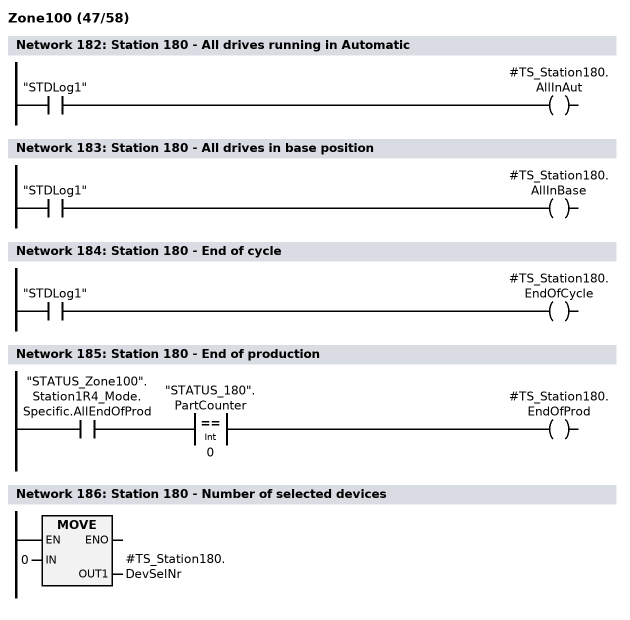
   RUNG wire#powerrail
      Contact( "STDLog1" )
      Coil( #TS_Station180.AllInAut )
   END_RUNG
   // the same network as SCL:
   #TS_Station180.AllInAut := "STDLog1";
END_REGION

REGION Network 183: Station 180 - All drives in base position
   RUNG wire#powerrail
      Contact( "STDLog1" )
      Coil( #TS_Station180.AllInBase )
   END_RUNG
   // the same network as SCL:
   #TS_Station180.AllInBase := "STDLog1";
END_REGION

REGION Network 184: Station 180 - End of cycle
   RUNG wire#powerrail
      Contact( "STDLog1" )
      Coil( #TS_Station180.EndOfCycle )
   END_RUNG
   // the same network as SCL:
   #TS_Station180.EndOfCycle := "STDLog1";
END_REGION

REGION Network 185: Station 180 - End of production
   RUNG wire#powerrail
      Contact( "STATUS_Zone100".Station1R4_Mode.Specific.AllEndOfProd )
      { S7_Templates := "SrcType := Int" } EQ_Contact(in1 := "STATUS_180".PartCounter, in2 := 0)
      Coil( #TS_Station180.EndOfProd )
   END_RUNG
   // the same network as SCL:
   #TS_Station180.EndOfProd := "STATUS_Zone100".Station1R4_Mode.Specific.AllEndOfProd AND ("STATUS_180".PartCounter = 0);
END_REGION

REGION Network 186: Station 180 - Number of selected devices
   RUNG wire#powerrail
      Move(in := 0, out1 => #TS_Station180.DevSelNr)
   END_RUNG
   // the same network as SCL:
   #TS_Station180.DevSelNr := 0;
END_REGION

REGION Network 187: Station 180 - Main control
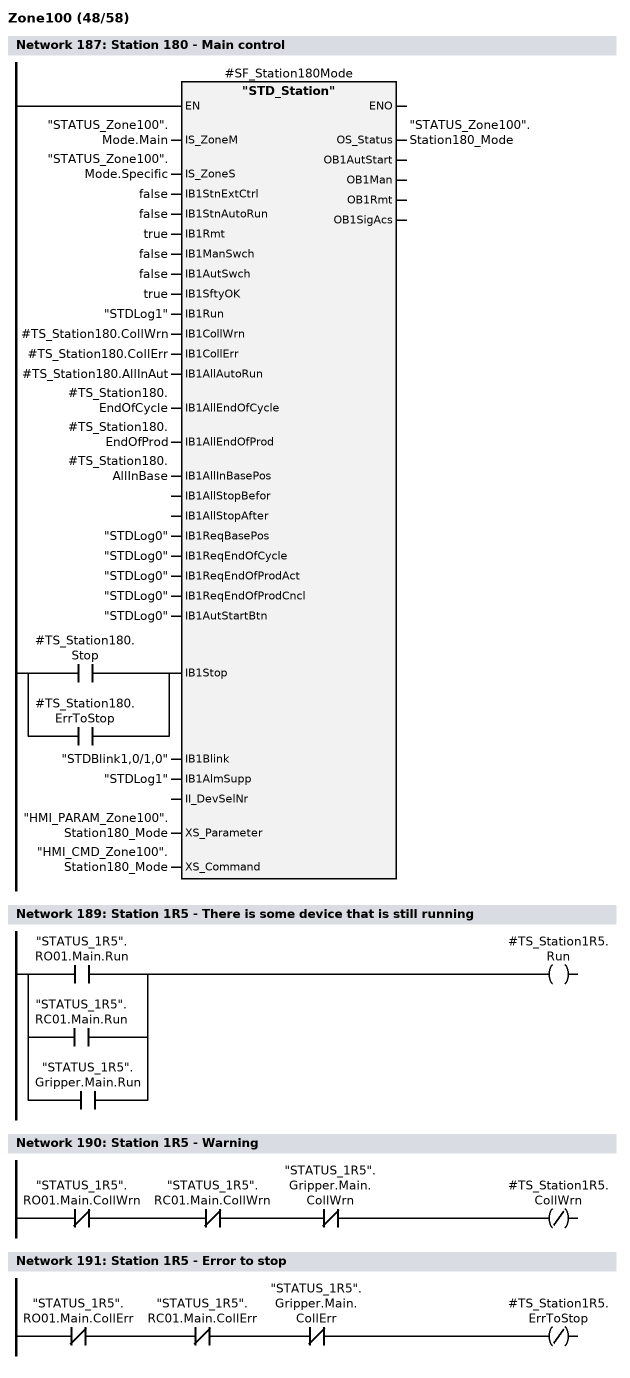
   RUNG wire#powerrail
      #SF_Station180Mode(IB1Stop := wire#w1, IS_ZoneM := "STATUS_Zone100".Mode.Main, IS_ZoneS := "STATUS_Zone100".Mode.Specific, IB1StnExtCtrl := false, IB1StnAutoRun := false, IB1Rmt := true, IB1ManSwch := false, IB1AutSwch := false, IB1SftyOK := true, IB1Run := "STDLog1", IB1CollWrn := #TS_Station180.CollWrn, IB1CollErr := #TS_Station180.CollErr, IB1AllAutoRun := #TS_Station180.AllInAut, IB1AllEndOfCycle := #TS_Station180.EndOfCycle, IB1AllEndOfProd := #TS_Station180.EndOfProd, IB1AllInBasePos := #TS_Station180.AllInBase, IB1AllStopBefor :=, IB1AllStopAfter :=, IB1ReqBasePos := "STDLog0", IB1ReqEndOfCycle := "STDLog0", IB1ReqEndOfProdAct := "STDLog0", IB1ReqEndOfProdCncl := "STDLog0", IB1AutStartBtn := "STDLog0", IB1Blink := "STDBlink1,0/1,0", IB1AlmSupp := "STDLog1", II_DevSelNr :=, XS_Parameter := "HMI_PARAM_Zone100".Station180_Mode, XS_Command := "HMI_CMD_Zone100".Station180_Mode, OS_Status => "STATUS_Zone100".Station180_Mode, OB1AutStart =>, OB1Man =>, OB1Rmt =>, OB1SigAcs =>)
   END_RUNG
   RUNG wire#powerrail
      Contact( #TS_Station180.Stop )
   END_RUNG wire#w1
   RUNG wire#powerrail
      Contact( #TS_Station180.ErrToStop )
   END_RUNG wire#w1
   // the same network as SCL:
   #SF_Station180Mode(IS_ZoneM := "STATUS_Zone100".Mode.Main,   // "STD_Station"
                      IS_ZoneS := "STATUS_Zone100".Mode.Specific,
                      IB1StnExtCtrl := false,
                      IB1StnAutoRun := false,
                      IB1Rmt := true,
                      IB1ManSwch := false,
                      IB1AutSwch := false,
                      IB1SftyOK := true,
                      IB1Run := "STDLog1",
                      IB1CollWrn := #TS_Station180.CollWrn,
                      IB1CollErr := #TS_Station180.CollErr,
                      IB1AllAutoRun := #TS_Station180.AllInAut,
                      IB1AllEndOfCycle := #TS_Station180.EndOfCycle,
                      IB1AllEndOfProd := #TS_Station180.EndOfProd,
                      IB1AllInBasePos := #TS_Station180.AllInBase,
                      IB1ReqBasePos := "STDLog0",
                      IB1ReqEndOfCycle := "STDLog0",
                      IB1ReqEndOfProdAct := "STDLog0",
                      IB1ReqEndOfProdCncl := "STDLog0",
                      IB1AutStartBtn := "STDLog0",
                      IB1Stop := #TS_Station180.Stop OR #TS_Station180.ErrToStop,
                      IB1Blink := "STDBlink1,0/1,0",
                      IB1AlmSupp := "STDLog1",
                      XS_Parameter := "HMI_PARAM_Zone100".Station180_Mode,
                      XS_Command := "HMI_CMD_Zone100".Station180_Mode,
                      OS_Status => "STATUS_Zone100".Station180_Mode);
END_REGION

REGION Network 188: *************** Station 1R5 ***************
END_REGION

REGION Network 189: Station 1R5 - There is some device that is still running
   RUNG wire#powerrail
      Contact( "STATUS_1R5".RO01.Main.Run )
      wire#w1
      Coil( #TS_Station1R5.Run )
   END_RUNG
   RUNG wire#powerrail
      Contact( "STATUS_1R5".RC01.Main.Run )
   END_RUNG wire#w1
   RUNG wire#powerrail
      Contact( "STATUS_1R5".Gripper.Main.Run )
   END_RUNG wire#w1
   // the same network as SCL:
   #TS_Station1R5.Run := "STATUS_1R5".RO01.Main.Run OR "STATUS_1R5".RC01.Main.Run OR "STATUS_1R5".Gripper.Main.Run;
END_REGION

REGION Network 190: Station 1R5 - Warning
   RUNG wire#powerrail
      I_Contact( "STATUS_1R5".RO01.Main.CollWrn )
      I_Contact( "STATUS_1R5".RC01.Main.CollWrn )
      I_Contact( "STATUS_1R5".Gripper.Main.CollWrn )
      I_Coil( #TS_Station1R5.CollWrn )
   END_RUNG
   // the same network as SCL:
   #TS_Station1R5.CollWrn := NOT (NOT "STATUS_1R5".RO01.Main.CollWrn AND NOT "STATUS_1R5".RC01.Main.CollWrn AND NOT "STATUS_1R5".Gripper.Main.CollWrn);
END_REGION

REGION Network 191: Station 1R5 - Error to stop
   RUNG wire#powerrail
      I_Contact( "STATUS_1R5".RO01.Main.CollErr )
      I_Contact( "STATUS_1R5".RC01.Main.CollErr )
      I_Contact( "STATUS_1R5".Gripper.Main.CollErr )
      I_Coil( #TS_Station1R5.ErrToStop )
   END_RUNG
   // the same network as SCL:
   #TS_Station1R5.ErrToStop := NOT (NOT "STATUS_1R5".RO01.Main.CollErr AND NOT "STATUS_1R5".RC01.Main.CollErr AND NOT "STATUS_1R5".Gripper.Main.CollErr);
END_REGION

REGION Network 192: Station 1R5 - Error (HMI purpose)
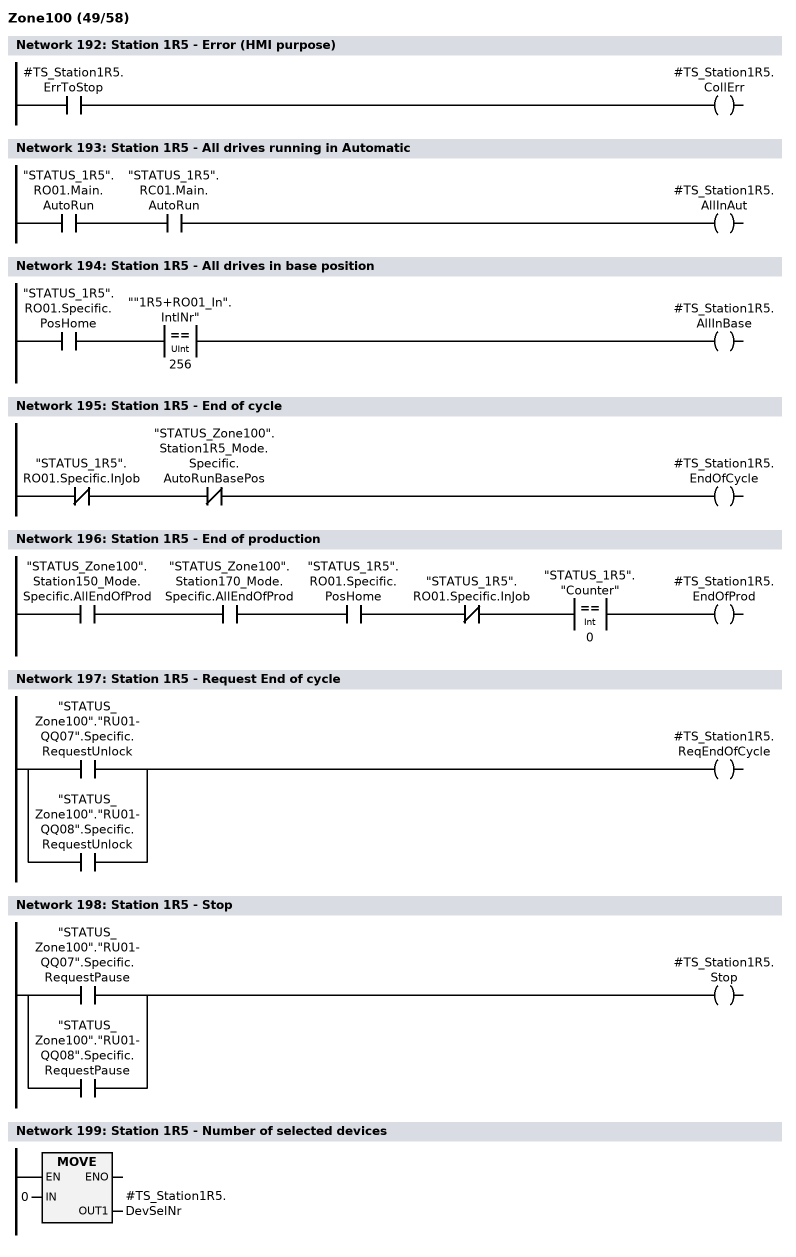
   RUNG wire#powerrail
      Contact( #TS_Station1R5.ErrToStop )
      Coil( #TS_Station1R5.CollErr )
   END_RUNG
   // the same network as SCL:
   #TS_Station1R5.CollErr := #TS_Station1R5.ErrToStop;
END_REGION

REGION Network 193: Station 1R5 - All drives running in Automatic
   RUNG wire#powerrail
      Contact( "STATUS_1R5".RO01.Main.AutoRun )
      Contact( "STATUS_1R5".RC01.Main.AutoRun )
      Coil( #TS_Station1R5.AllInAut )
   END_RUNG
   // the same network as SCL:
   #TS_Station1R5.AllInAut := "STATUS_1R5".RO01.Main.AutoRun AND "STATUS_1R5".RC01.Main.AutoRun;
END_REGION

REGION Network 194: Station 1R5 - All drives in base position
   RUNG wire#powerrail
      Contact( "STATUS_1R5".RO01.Specific.PosHome )
      { S7_Templates := "SrcType := UInt" } EQ_Contact(in1 := ""1R5+RO01_In".IntlNr", in2 := 256)
      Coil( #TS_Station1R5.AllInBase )
   END_RUNG
   // the same network as SCL:
   // no checked SCL form for this network; see the picture
END_REGION

REGION Network 195: Station 1R5 - End of cycle
   RUNG wire#powerrail
      I_Contact( "STATUS_1R5".RO01.Specific.InJob )
      I_Contact( "STATUS_Zone100".Station1R5_Mode.Specific.AutoRunBasePos )
      Coil( #TS_Station1R5.EndOfCycle )
   END_RUNG
   // the same network as SCL:
   #TS_Station1R5.EndOfCycle := NOT "STATUS_1R5".RO01.Specific.InJob AND NOT "STATUS_Zone100".Station1R5_Mode.Specific.AutoRunBasePos;
END_REGION

REGION Network 196: Station 1R5 - End of production
   RUNG wire#powerrail
      Contact( "STATUS_Zone100".Station150_Mode.Specific.AllEndOfProd )
      Contact( "STATUS_Zone100".Station170_Mode.Specific.AllEndOfProd )
      Contact( "STATUS_1R5".RO01.Specific.PosHome )
      I_Contact( "STATUS_1R5".RO01.Specific.InJob )
      { S7_Templates := "SrcType := Int" } EQ_Contact(in1 := "STATUS_1R5"."Counter", in2 := 0)
      Coil( #TS_Station1R5.EndOfProd )
   END_RUNG
   // the same network as SCL:
   #TS_Station1R5.EndOfProd := "STATUS_Zone100".Station150_Mode.Specific.AllEndOfProd AND "STATUS_Zone100".Station170_Mode.Specific.AllEndOfProd AND "STATUS_1R5".RO01.Specific.PosHome AND NOT "STATUS_1R5".RO01.Specific.InJob AND ("STATUS_1R5"."Counter" = 0);
END_REGION

REGION Network 197: Station 1R5 - Request End of cycle
   RUNG wire#powerrail
      Contact( "STATUS_Zone100"."RU01-QQ07".Specific.RequestUnlock )
      wire#w1
      Coil( #TS_Station1R5.ReqEndOfCycle )
   END_RUNG
   RUNG wire#powerrail
      Contact( "STATUS_Zone100"."RU01-QQ08".Specific.RequestUnlock )
   END_RUNG wire#w1
   // the same network as SCL:
   #TS_Station1R5.ReqEndOfCycle := "STATUS_Zone100"."RU01-QQ07".Specific.RequestUnlock OR "STATUS_Zone100"."RU01-QQ08".Specific.RequestUnlock;
END_REGION

REGION Network 198: Station 1R5 - Stop
   RUNG wire#powerrail
      Contact( "STATUS_Zone100"."RU01-QQ07".Specific.RequestPause )
      wire#w1
      Coil( #TS_Station1R5.Stop )
   END_RUNG
   RUNG wire#powerrail
      Contact( "STATUS_Zone100"."RU01-QQ08".Specific.RequestPause )
   END_RUNG wire#w1
   // the same network as SCL:
   #TS_Station1R5.Stop := "STATUS_Zone100"."RU01-QQ07".Specific.RequestPause OR "STATUS_Zone100"."RU01-QQ08".Specific.RequestPause;
END_REGION

REGION Network 199: Station 1R5 - Number of selected devices
   RUNG wire#powerrail
      Move(in := 0, out1 => #TS_Station1R5.DevSelNr)
   END_RUNG
   // the same network as SCL:
   #TS_Station1R5.DevSelNr := 0;
END_REGION

REGION Network 200: Station 1R5 - AutoOn edges
   // Its needed for #SB1ModeOff in STD_Station block
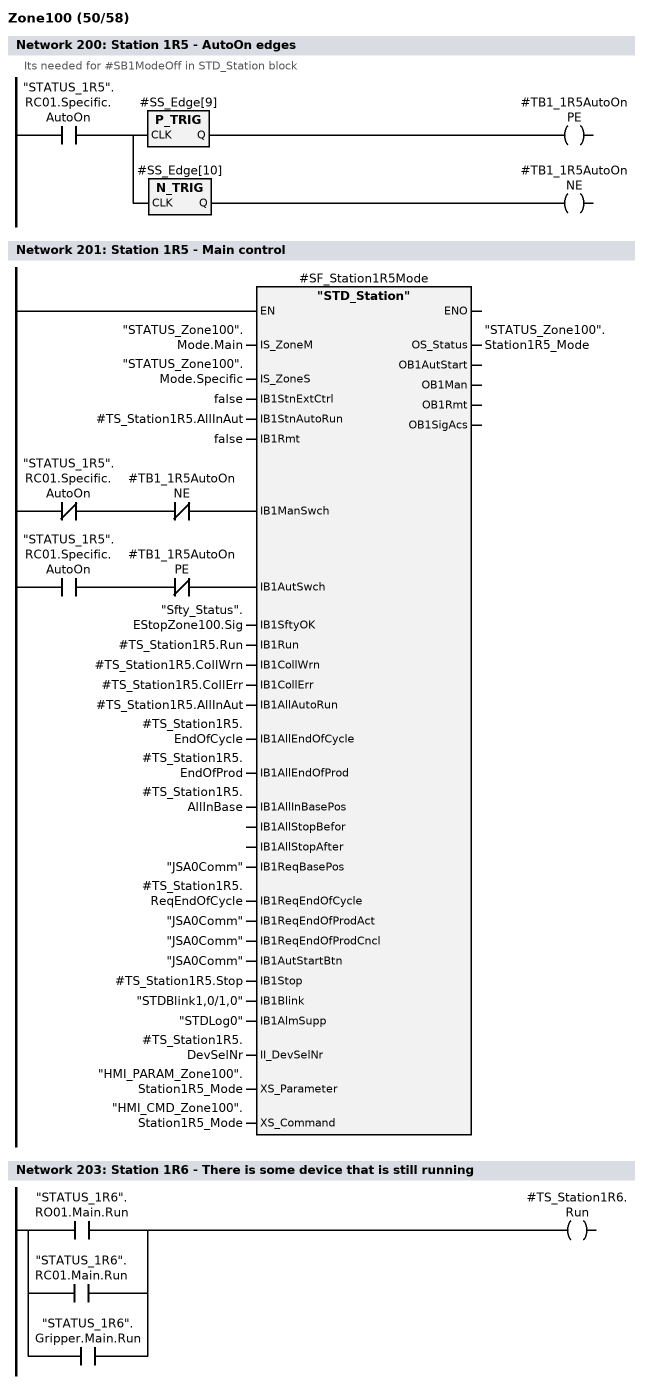
   RUNG wire#powerrail
      Contact( "STATUS_1R5".RC01.Specific.AutoOn )
      wire#w1
      P_Trig( #SS_Edge[9] )
      Coil( #TB1_1R5AutoOnPE )
   END_RUNG
   RUNG wire#w1
      N_Trig( #SS_Edge[10] )
      Coil( #TB1_1R5AutoOnNE )
   END_RUNG
   // the same network as SCL:
   #_w1 := "STATUS_1R5".RC01.Specific.AutoOn AND NOT #SS_Edge[9];   // rising edge
   #SS_Edge[9] := "STATUS_1R5".RC01.Specific.AutoOn;
   #TB1_1R5AutoOnPE := #_w1;
   #_w2 := NOT "STATUS_1R5".RC01.Specific.AutoOn AND #SS_Edge[10];   // falling edge
   #SS_Edge[10] := "STATUS_1R5".RC01.Specific.AutoOn;
   #TB1_1R5AutoOnNE := #_w2;
END_REGION

REGION Network 201: Station 1R5 - Main control
   RUNG wire#powerrail
      #SF_Station1R5Mode(IB1ManSwch := wire#w1, IB1AutSwch := wire#w2, IS_ZoneM := "STATUS_Zone100".Mode.Main, IS_ZoneS := "STATUS_Zone100".Mode.Specific, IB1StnExtCtrl := false, IB1StnAutoRun := #TS_Station1R5.AllInAut, IB1Rmt := false, IB1SftyOK := "Sfty_Status".EStopZone100.Sig, IB1Run := #TS_Station1R5.Run, IB1CollWrn := #TS_Station1R5.CollWrn, IB1CollErr := #TS_Station1R5.CollErr, IB1AllAutoRun := #TS_Station1R5.AllInAut, IB1AllEndOfCycle := #TS_Station1R5.EndOfCycle, IB1AllEndOfProd := #TS_Station1R5.EndOfProd, IB1AllInBasePos := #TS_Station1R5.AllInBase, IB1AllStopBefor :=, IB1AllStopAfter :=, IB1ReqBasePos := "JSA0Comm", IB1ReqEndOfCycle := #TS_Station1R5.ReqEndOfCycle, IB1ReqEndOfProdAct := "JSA0Comm", IB1ReqEndOfProdCncl := "JSA0Comm", IB1AutStartBtn := "JSA0Comm", IB1Stop := #TS_Station1R5.Stop, IB1Blink := "STDBlink1,0/1,0", IB1AlmSupp := "STDLog0", II_DevSelNr := #TS_Station1R5.DevSelNr, XS_Parameter := "HMI_PARAM_Zone100".Station1R5_Mode, XS_Command := "HMI_CMD_Zone100".Station1R5_Mode, OS_Status => "STATUS_Zone100".Station1R5_Mode, OB1AutStart =>, OB1Man =>, OB1Rmt =>, OB1SigAcs =>)
   END_RUNG
   RUNG wire#powerrail
      I_Contact( "STATUS_1R5".RC01.Specific.AutoOn )
      I_Contact( #TB1_1R5AutoOnNE )
   END_RUNG wire#w1
   RUNG wire#powerrail
      Contact( "STATUS_1R5".RC01.Specific.AutoOn )
      I_Contact( #TB1_1R5AutoOnPE )
   END_RUNG wire#w2
   // the same network as SCL:
   #SF_Station1R5Mode(IS_ZoneM := "STATUS_Zone100".Mode.Main,   // "STD_Station"
                      IS_ZoneS := "STATUS_Zone100".Mode.Specific,
                      IB1StnExtCtrl := false,
                      IB1StnAutoRun := #TS_Station1R5.AllInAut,
                      IB1Rmt := false,
                      IB1ManSwch := NOT "STATUS_1R5".RC01.Specific.AutoOn AND NOT #TB1_1R5AutoOnNE,
                      IB1AutSwch := "STATUS_1R5".RC01.Specific.AutoOn AND NOT #TB1_1R5AutoOnPE,
                      IB1SftyOK := "Sfty_Status".EStopZone100.Sig,
                      IB1Run := #TS_Station1R5.Run,
                      IB1CollWrn := #TS_Station1R5.CollWrn,
                      IB1CollErr := #TS_Station1R5.CollErr,
                      IB1AllAutoRun := #TS_Station1R5.AllInAut,
                      IB1AllEndOfCycle := #TS_Station1R5.EndOfCycle,
                      IB1AllEndOfProd := #TS_Station1R5.EndOfProd,
                      IB1AllInBasePos := #TS_Station1R5.AllInBase,
                      IB1ReqBasePos := "JSA0Comm",
                      IB1ReqEndOfCycle := #TS_Station1R5.ReqEndOfCycle,
                      IB1ReqEndOfProdAct := "JSA0Comm",
                      IB1ReqEndOfProdCncl := "JSA0Comm",
                      IB1AutStartBtn := "JSA0Comm",
                      IB1Stop := #TS_Station1R5.Stop,
                      IB1Blink := "STDBlink1,0/1,0",
                      IB1AlmSupp := "STDLog0",
                      II_DevSelNr := #TS_Station1R5.DevSelNr,
                      XS_Parameter := "HMI_PARAM_Zone100".Station1R5_Mode,
                      XS_Command := "HMI_CMD_Zone100".Station1R5_Mode,
                      OS_Status => "STATUS_Zone100".Station1R5_Mode);
END_REGION

REGION Network 202: *************** Station 1R6 ***************
END_REGION

REGION Network 203: Station 1R6 - There is some device that is still running
   RUNG wire#powerrail
      Contact( "STATUS_1R6".RO01.Main.Run )
      wire#w1
      Coil( #TS_Station1R6.Run )
   END_RUNG
   RUNG wire#powerrail
      Contact( "STATUS_1R6".RC01.Main.Run )
   END_RUNG wire#w1
   RUNG wire#powerrail
      Contact( "STATUS_1R6".Gripper.Main.Run )
   END_RUNG wire#w1
   // the same network as SCL:
   #TS_Station1R6.Run := "STATUS_1R6".RO01.Main.Run OR "STATUS_1R6".RC01.Main.Run OR "STATUS_1R6".Gripper.Main.Run;
END_REGION

REGION Network 204: Station 1R6 - Warning
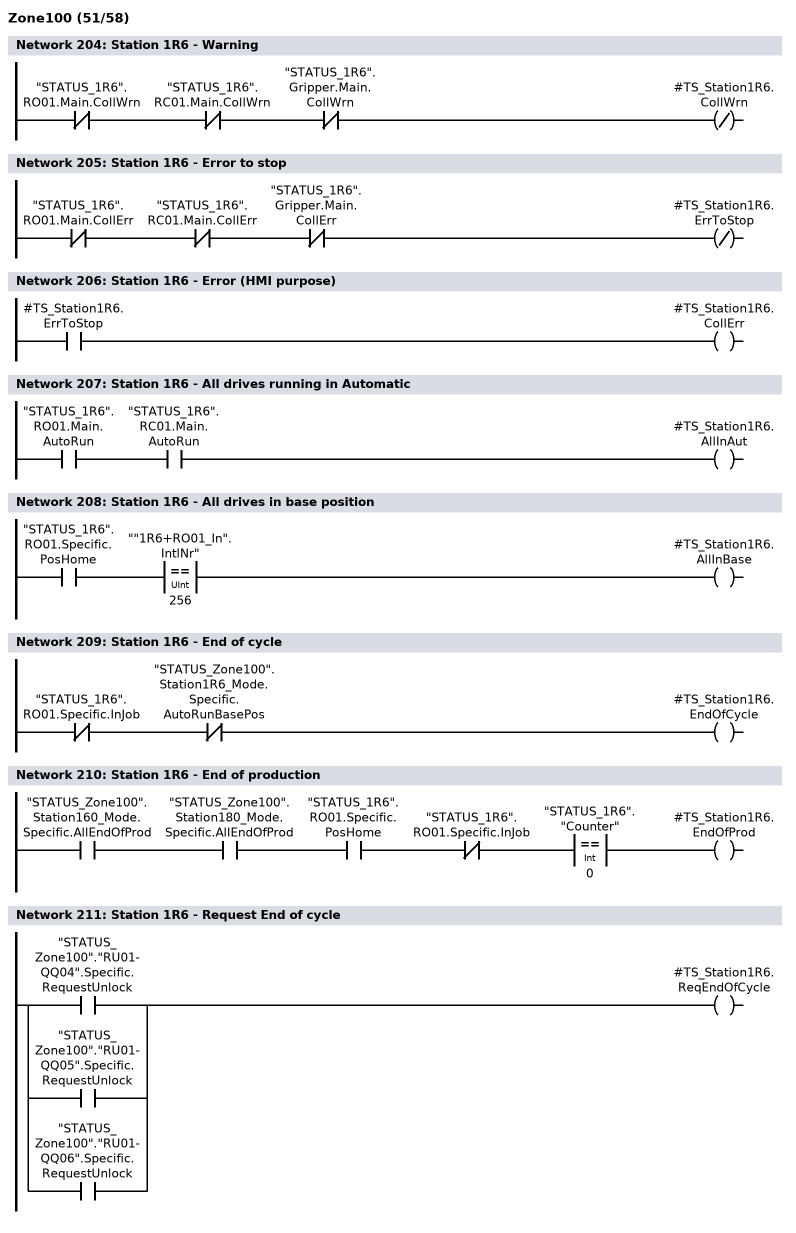
   RUNG wire#powerrail
      I_Contact( "STATUS_1R6".RO01.Main.CollWrn )
      I_Contact( "STATUS_1R6".RC01.Main.CollWrn )
      I_Contact( "STATUS_1R6".Gripper.Main.CollWrn )
      I_Coil( #TS_Station1R6.CollWrn )
   END_RUNG
   // the same network as SCL:
   #TS_Station1R6.CollWrn := NOT (NOT "STATUS_1R6".RO01.Main.CollWrn AND NOT "STATUS_1R6".RC01.Main.CollWrn AND NOT "STATUS_1R6".Gripper.Main.CollWrn);
END_REGION

REGION Network 205: Station 1R6 - Error to stop
   RUNG wire#powerrail
      I_Contact( "STATUS_1R6".RO01.Main.CollErr )
      I_Contact( "STATUS_1R6".RC01.Main.CollErr )
      I_Contact( "STATUS_1R6".Gripper.Main.CollErr )
      I_Coil( #TS_Station1R6.ErrToStop )
   END_RUNG
   // the same network as SCL:
   #TS_Station1R6.ErrToStop := NOT (NOT "STATUS_1R6".RO01.Main.CollErr AND NOT "STATUS_1R6".RC01.Main.CollErr AND NOT "STATUS_1R6".Gripper.Main.CollErr);
END_REGION

REGION Network 206: Station 1R6 - Error (HMI purpose)
   RUNG wire#powerrail
      Contact( #TS_Station1R6.ErrToStop )
      Coil( #TS_Station1R6.CollErr )
   END_RUNG
   // the same network as SCL:
   #TS_Station1R6.CollErr := #TS_Station1R6.ErrToStop;
END_REGION

REGION Network 207: Station 1R6 - All drives running in Automatic
   RUNG wire#powerrail
      Contact( "STATUS_1R6".RO01.Main.AutoRun )
      Contact( "STATUS_1R6".RC01.Main.AutoRun )
      Coil( #TS_Station1R6.AllInAut )
   END_RUNG
   // the same network as SCL:
   #TS_Station1R6.AllInAut := "STATUS_1R6".RO01.Main.AutoRun AND "STATUS_1R6".RC01.Main.AutoRun;
END_REGION

REGION Network 208: Station 1R6 - All drives in base position
   RUNG wire#powerrail
      Contact( "STATUS_1R6".RO01.Specific.PosHome )
      { S7_Templates := "SrcType := UInt" } EQ_Contact(in1 := ""1R6+RO01_In".IntlNr", in2 := 256)
      Coil( #TS_Station1R6.AllInBase )
   END_RUNG
   // the same network as SCL:
   // no checked SCL form for this network; see the picture
END_REGION

REGION Network 209: Station 1R6 - End of cycle
   RUNG wire#powerrail
      I_Contact( "STATUS_1R6".RO01.Specific.InJob )
      I_Contact( "STATUS_Zone100".Station1R6_Mode.Specific.AutoRunBasePos )
      Coil( #TS_Station1R6.EndOfCycle )
   END_RUNG
   // the same network as SCL:
   #TS_Station1R6.EndOfCycle := NOT "STATUS_1R6".RO01.Specific.InJob AND NOT "STATUS_Zone100".Station1R6_Mode.Specific.AutoRunBasePos;
END_REGION

REGION Network 210: Station 1R6 - End of production
   RUNG wire#powerrail
      Contact( "STATUS_Zone100".Station160_Mode.Specific.AllEndOfProd )
      Contact( "STATUS_Zone100".Station180_Mode.Specific.AllEndOfProd )
      Contact( "STATUS_1R6".RO01.Specific.PosHome )
      I_Contact( "STATUS_1R6".RO01.Specific.InJob )
      { S7_Templates := "SrcType := Int" } EQ_Contact(in1 := "STATUS_1R6"."Counter", in2 := 0)
      Coil( #TS_Station1R6.EndOfProd )
   END_RUNG
   // the same network as SCL:
   #TS_Station1R6.EndOfProd := "STATUS_Zone100".Station160_Mode.Specific.AllEndOfProd AND "STATUS_Zone100".Station180_Mode.Specific.AllEndOfProd AND "STATUS_1R6".RO01.Specific.PosHome AND NOT "STATUS_1R6".RO01.Specific.InJob AND ("STATUS_1R6"."Counter" = 0);
END_REGION

REGION Network 211: Station 1R6 - Request End of cycle
   RUNG wire#powerrail
      Contact( "STATUS_Zone100"."RU01-QQ04".Specific.RequestUnlock )
      wire#w1
      Coil( #TS_Station1R6.ReqEndOfCycle )
   END_RUNG
   RUNG wire#powerrail
      Contact( "STATUS_Zone100"."RU01-QQ05".Specific.RequestUnlock )
   END_RUNG wire#w1
   RUNG wire#powerrail
      Contact( "STATUS_Zone100"."RU01-QQ06".Specific.RequestUnlock )
   END_RUNG wire#w1
   // the same network as SCL:
   #TS_Station1R6.ReqEndOfCycle := "STATUS_Zone100"."RU01-QQ04".Specific.RequestUnlock OR "STATUS_Zone100"."RU01-QQ05".Specific.RequestUnlock OR "STATUS_Zone100"."RU01-QQ06".Specific.RequestUnlock;
END_REGION

REGION Network 212: Station 1R6 - Stop
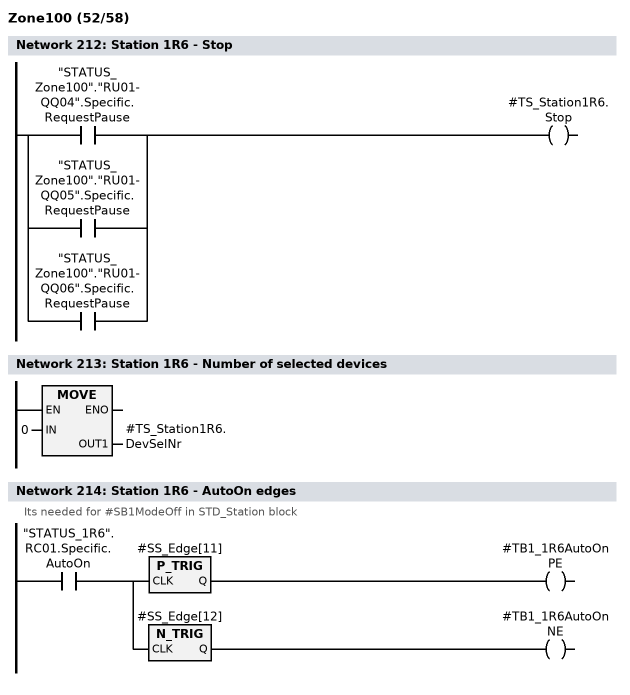
   RUNG wire#powerrail
      Contact( "STATUS_Zone100"."RU01-QQ04".Specific.RequestPause )
      wire#w1
      Coil( #TS_Station1R6.Stop )
   END_RUNG
   RUNG wire#powerrail
      Contact( "STATUS_Zone100"."RU01-QQ05".Specific.RequestPause )
   END_RUNG wire#w1
   RUNG wire#powerrail
      Contact( "STATUS_Zone100"."RU01-QQ06".Specific.RequestPause )
   END_RUNG wire#w1
   // the same network as SCL:
   #TS_Station1R6.Stop := "STATUS_Zone100"."RU01-QQ04".Specific.RequestPause OR "STATUS_Zone100"."RU01-QQ05".Specific.RequestPause OR "STATUS_Zone100"."RU01-QQ06".Specific.RequestPause;
END_REGION

REGION Network 213: Station 1R6 - Number of selected devices
   RUNG wire#powerrail
      Move(in := 0, out1 => #TS_Station1R6.DevSelNr)
   END_RUNG
   // the same network as SCL:
   #TS_Station1R6.DevSelNr := 0;
END_REGION

REGION Network 214: Station 1R6 - AutoOn edges
   // Its needed for #SB1ModeOff in STD_Station block
   RUNG wire#powerrail
      Contact( "STATUS_1R6".RC01.Specific.AutoOn )
      wire#w1
      P_Trig( #SS_Edge[11] )
      Coil( #TB1_1R6AutoOnPE )
   END_RUNG
   RUNG wire#w1
      N_Trig( #SS_Edge[12] )
      Coil( #TB1_1R6AutoOnNE )
   END_RUNG
   // the same network as SCL:
   #_w1 := "STATUS_1R6".RC01.Specific.AutoOn AND NOT #SS_Edge[11];   // rising edge
   #SS_Edge[11] := "STATUS_1R6".RC01.Specific.AutoOn;
   #TB1_1R6AutoOnPE := #_w1;
   #_w2 := NOT "STATUS_1R6".RC01.Specific.AutoOn AND #SS_Edge[12];   // falling edge
   #SS_Edge[12] := "STATUS_1R6".RC01.Specific.AutoOn;
   #TB1_1R6AutoOnNE := #_w2;
END_REGION

REGION Network 215: Station 1R6 - Main control
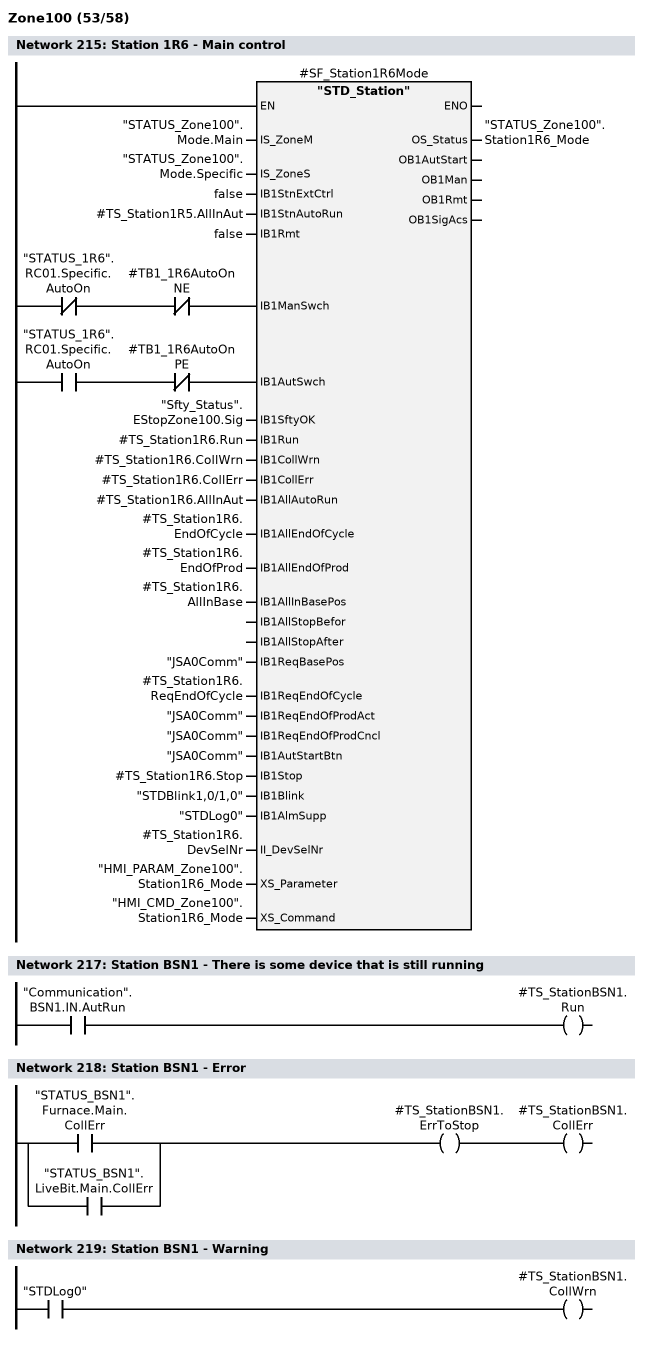
   RUNG wire#powerrail
      #SF_Station1R6Mode(IB1ManSwch := wire#w1, IB1AutSwch := wire#w2, IS_ZoneM := "STATUS_Zone100".Mode.Main, IS_ZoneS := "STATUS_Zone100".Mode.Specific, IB1StnExtCtrl := false, IB1StnAutoRun := #TS_Station1R5.AllInAut, IB1Rmt := false, IB1SftyOK := "Sfty_Status".EStopZone100.Sig, IB1Run := #TS_Station1R6.Run, IB1CollWrn := #TS_Station1R6.CollWrn, IB1CollErr := #TS_Station1R6.CollErr, IB1AllAutoRun := #TS_Station1R6.AllInAut, IB1AllEndOfCycle := #TS_Station1R6.EndOfCycle, IB1AllEndOfProd := #TS_Station1R6.EndOfProd, IB1AllInBasePos := #TS_Station1R6.AllInBase, IB1AllStopBefor :=, IB1AllStopAfter :=, IB1ReqBasePos := "JSA0Comm", IB1ReqEndOfCycle := #TS_Station1R6.ReqEndOfCycle, IB1ReqEndOfProdAct := "JSA0Comm", IB1ReqEndOfProdCncl := "JSA0Comm", IB1AutStartBtn := "JSA0Comm", IB1Stop := #TS_Station1R6.Stop, IB1Blink := "STDBlink1,0/1,0", IB1AlmSupp := "STDLog0", II_DevSelNr := #TS_Station1R6.DevSelNr, XS_Parameter := "HMI_PARAM_Zone100".Station1R6_Mode, XS_Command := "HMI_CMD_Zone100".Station1R6_Mode, OS_Status => "STATUS_Zone100".Station1R6_Mode, OB1AutStart =>, OB1Man =>, OB1Rmt =>, OB1SigAcs =>)
   END_RUNG
   RUNG wire#powerrail
      I_Contact( "STATUS_1R6".RC01.Specific.AutoOn )
      I_Contact( #TB1_1R6AutoOnNE )
   END_RUNG wire#w1
   RUNG wire#powerrail
      Contact( "STATUS_1R6".RC01.Specific.AutoOn )
      I_Contact( #TB1_1R6AutoOnPE )
   END_RUNG wire#w2
   // the same network as SCL:
   #SF_Station1R6Mode(IS_ZoneM := "STATUS_Zone100".Mode.Main,   // "STD_Station"
                      IS_ZoneS := "STATUS_Zone100".Mode.Specific,
                      IB1StnExtCtrl := false,
                      IB1StnAutoRun := #TS_Station1R5.AllInAut,
                      IB1Rmt := false,
                      IB1ManSwch := NOT "STATUS_1R6".RC01.Specific.AutoOn AND NOT #TB1_1R6AutoOnNE,
                      IB1AutSwch := "STATUS_1R6".RC01.Specific.AutoOn AND NOT #TB1_1R6AutoOnPE,
                      IB1SftyOK := "Sfty_Status".EStopZone100.Sig,
                      IB1Run := #TS_Station1R6.Run,
                      IB1CollWrn := #TS_Station1R6.CollWrn,
                      IB1CollErr := #TS_Station1R6.CollErr,
                      IB1AllAutoRun := #TS_Station1R6.AllInAut,
                      IB1AllEndOfCycle := #TS_Station1R6.EndOfCycle,
                      IB1AllEndOfProd := #TS_Station1R6.EndOfProd,
                      IB1AllInBasePos := #TS_Station1R6.AllInBase,
                      IB1ReqBasePos := "JSA0Comm",
                      IB1ReqEndOfCycle := #TS_Station1R6.ReqEndOfCycle,
                      IB1ReqEndOfProdAct := "JSA0Comm",
                      IB1ReqEndOfProdCncl := "JSA0Comm",
                      IB1AutStartBtn := "JSA0Comm",
                      IB1Stop := #TS_Station1R6.Stop,
                      IB1Blink := "STDBlink1,0/1,0",
                      IB1AlmSupp := "STDLog0",
                      II_DevSelNr := #TS_Station1R6.DevSelNr,
                      XS_Parameter := "HMI_PARAM_Zone100".Station1R6_Mode,
                      XS_Command := "HMI_CMD_Zone100".Station1R6_Mode,
                      OS_Status => "STATUS_Zone100".Station1R6_Mode);
END_REGION

REGION Network 216: *************** Station BSN1 ***************
END_REGION

REGION Network 217: Station BSN1 - There is some device that is still running
   RUNG wire#powerrail
      Contact( "Communication".BSN1.IN.AutRun )
      Coil( #TS_StationBSN1.Run )
   END_RUNG
   // the same network as SCL:
   #TS_StationBSN1.Run := "Communication".BSN1.IN.AutRun;
END_REGION

REGION Network 218: Station BSN1 - Error
   RUNG wire#powerrail
      Contact( "STATUS_BSN1".Furnace.Main.CollErr )
      wire#w1
      Coil( #TS_StationBSN1.ErrToStop )
      Coil( #TS_StationBSN1.CollErr )
   END_RUNG
   RUNG wire#powerrail
      Contact( "STATUS_BSN1".LiveBit.Main.CollErr )
   END_RUNG wire#w1
   // the same network as SCL:
   #TS_StationBSN1.ErrToStop := "STATUS_BSN1".Furnace.Main.CollErr OR "STATUS_BSN1".LiveBit.Main.CollErr;
   #TS_StationBSN1.CollErr := #TS_StationBSN1.ErrToStop;
END_REGION

REGION Network 219: Station BSN1 - Warning
   RUNG wire#powerrail
      Contact( "STDLog0" )
      Coil( #TS_StationBSN1.CollWrn )
   END_RUNG
   // the same network as SCL:
   #TS_StationBSN1.CollWrn := "STDLog0";
END_REGION

REGION Network 220: Station BSN1 - All drives running in Automatic
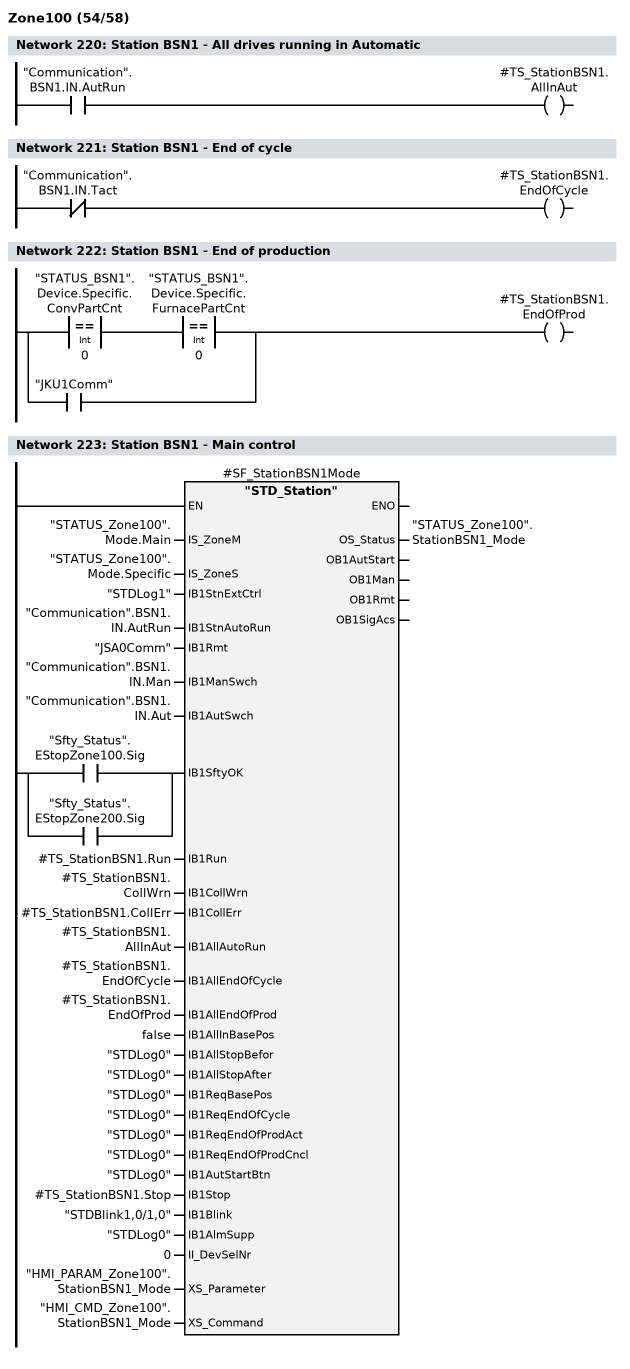
   RUNG wire#powerrail
      Contact( "Communication".BSN1.IN.AutRun )
      Coil( #TS_StationBSN1.AllInAut )
   END_RUNG
   // the same network as SCL:
   #TS_StationBSN1.AllInAut := "Communication".BSN1.IN.AutRun;
END_REGION

REGION Network 221: Station BSN1 - End of cycle
   RUNG wire#powerrail
      I_Contact( "Communication".BSN1.IN.Tact )
      Coil( #TS_StationBSN1.EndOfCycle )
   END_RUNG
   // the same network as SCL:
   #TS_StationBSN1.EndOfCycle := NOT "Communication".BSN1.IN.Tact;
END_REGION

REGION Network 222: Station BSN1 - End of production
   RUNG wire#powerrail
      { S7_Templates := "SrcType := Int" } EQ_Contact(in1 := "STATUS_BSN1".Device.Specific.ConvPartCnt, in2 := 0)
      { S7_Templates := "SrcType := Int" } EQ_Contact(in1 := "STATUS_BSN1".Device.Specific.FurnacePartCnt, in2 := 0)
      wire#w1
      Coil( #TS_StationBSN1.EndOfProd )
   END_RUNG
   RUNG wire#powerrail
      Contact( "JKU1Comm" )
   END_RUNG wire#w1
   // the same network as SCL:
   #TS_StationBSN1.EndOfProd := (("STATUS_BSN1".Device.Specific.ConvPartCnt = 0) AND ("STATUS_BSN1".Device.Specific.FurnacePartCnt = 0)) OR "JKU1Comm";
END_REGION

REGION Network 223: Station BSN1 - Main control
   RUNG wire#powerrail
      #SF_StationBSN1Mode(IB1SftyOK := wire#w1, IS_ZoneM := "STATUS_Zone100".Mode.Main, IS_ZoneS := "STATUS_Zone100".Mode.Specific, IB1StnExtCtrl := "STDLog1", IB1StnAutoRun := "Communication".BSN1.IN.AutRun, IB1Rmt := "JSA0Comm", IB1ManSwch := "Communication".BSN1.IN.Man, IB1AutSwch := "Communication".BSN1.IN.Aut, IB1Run := #TS_StationBSN1.Run, IB1CollWrn := #TS_StationBSN1.CollWrn, IB1CollErr := #TS_StationBSN1.CollErr, IB1AllAutoRun := #TS_StationBSN1.AllInAut, IB1AllEndOfCycle := #TS_StationBSN1.EndOfCycle, IB1AllEndOfProd := #TS_StationBSN1.EndOfProd, IB1AllInBasePos := false, IB1AllStopBefor := "STDLog0", IB1AllStopAfter := "STDLog0", IB1ReqBasePos := "STDLog0", IB1ReqEndOfCycle := "STDLog0", IB1ReqEndOfProdAct := "STDLog0", IB1ReqEndOfProdCncl := "STDLog0", IB1AutStartBtn := "STDLog0", IB1Stop := #TS_StationBSN1.Stop, IB1Blink := "STDBlink1,0/1,0", IB1AlmSupp := "STDLog0", II_DevSelNr := 0, XS_Parameter := "HMI_PARAM_Zone100".StationBSN1_Mode, XS_Command := "HMI_CMD_Zone100".StationBSN1_Mode, OS_Status => "STATUS_Zone100".StationBSN1_Mode, OB1AutStart =>, OB1Man =>, OB1Rmt =>, OB1SigAcs =>)
   END_RUNG
   RUNG wire#powerrail
      Contact( "Sfty_Status".EStopZone100.Sig )
   END_RUNG wire#w1
   RUNG wire#powerrail
      Contact( "Sfty_Status".EStopZone200.Sig )
   END_RUNG wire#w1
   // the same network as SCL:
   #SF_StationBSN1Mode(IS_ZoneM := "STATUS_Zone100".Mode.Main,   // "STD_Station"
                       IS_ZoneS := "STATUS_Zone100".Mode.Specific,
                       IB1StnExtCtrl := "STDLog1",
                       IB1StnAutoRun := "Communication".BSN1.IN.AutRun,
                       IB1Rmt := "JSA0Comm",
                       IB1ManSwch := "Communication".BSN1.IN.Man,
                       IB1AutSwch := "Communication".BSN1.IN.Aut,
                       IB1SftyOK := "Sfty_Status".EStopZone100.Sig OR "Sfty_Status".EStopZone200.Sig,
                       IB1Run := #TS_StationBSN1.Run,
                       IB1CollWrn := #TS_StationBSN1.CollWrn,
                       IB1CollErr := #TS_StationBSN1.CollErr,
                       IB1AllAutoRun := #TS_StationBSN1.AllInAut,
                       IB1AllEndOfCycle := #TS_StationBSN1.EndOfCycle,
                       IB1AllEndOfProd := #TS_StationBSN1.EndOfProd,
                       IB1AllInBasePos := false,
                       IB1AllStopBefor := "STDLog0",
                       IB1AllStopAfter := "STDLog0",
                       IB1ReqBasePos := "STDLog0",
                       IB1ReqEndOfCycle := "STDLog0",
                       IB1ReqEndOfProdAct := "STDLog0",
                       IB1ReqEndOfProdCncl := "STDLog0",
                       IB1AutStartBtn := "STDLog0",
                       IB1Stop := #TS_StationBSN1.Stop,
                       IB1Blink := "STDBlink1,0/1,0",
                       IB1AlmSupp := "STDLog0",
                       II_DevSelNr := 0,
                       XS_Parameter := "HMI_PARAM_Zone100".StationBSN1_Mode,
                       XS_Command := "HMI_CMD_Zone100".StationBSN1_Mode,
                       OS_Status => "STATUS_Zone100".StationBSN1_Mode);
END_REGION

REGION Network 224: *************** Station BSN2 ***************
END_REGION

REGION Network 225: Station BSN2 - There is some device that is still running
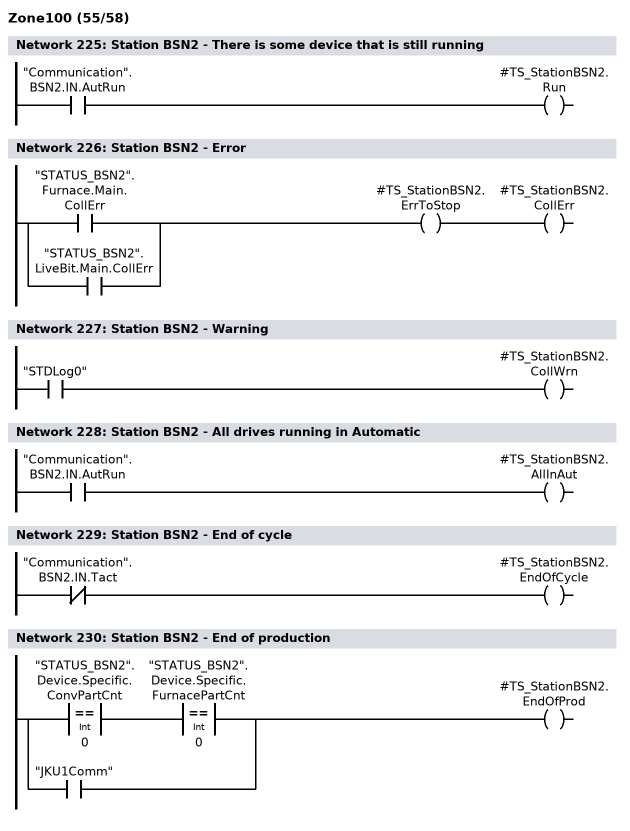
   RUNG wire#powerrail
      Contact( "Communication".BSN2.IN.AutRun )
      Coil( #TS_StationBSN2.Run )
   END_RUNG
   // the same network as SCL:
   #TS_StationBSN2.Run := "Communication".BSN2.IN.AutRun;
END_REGION

REGION Network 226: Station BSN2 - Error
   RUNG wire#powerrail
      Contact( "STATUS_BSN2".Furnace.Main.CollErr )
      wire#w1
      Coil( #TS_StationBSN2.ErrToStop )
      Coil( #TS_StationBSN2.CollErr )
   END_RUNG
   RUNG wire#powerrail
      Contact( "STATUS_BSN2".LiveBit.Main.CollErr )
   END_RUNG wire#w1
   // the same network as SCL:
   #TS_StationBSN2.ErrToStop := "STATUS_BSN2".Furnace.Main.CollErr OR "STATUS_BSN2".LiveBit.Main.CollErr;
   #TS_StationBSN2.CollErr := #TS_StationBSN2.ErrToStop;
END_REGION

REGION Network 227: Station BSN2 - Warning
   RUNG wire#powerrail
      Contact( "STDLog0" )
      Coil( #TS_StationBSN2.CollWrn )
   END_RUNG
   // the same network as SCL:
   #TS_StationBSN2.CollWrn := "STDLog0";
END_REGION

REGION Network 228: Station BSN2 - All drives running in Automatic
   RUNG wire#powerrail
      Contact( "Communication".BSN2.IN.AutRun )
      Coil( #TS_StationBSN2.AllInAut )
   END_RUNG
   // the same network as SCL:
   #TS_StationBSN2.AllInAut := "Communication".BSN2.IN.AutRun;
END_REGION

REGION Network 229: Station BSN2 - End of cycle
   RUNG wire#powerrail
      I_Contact( "Communication".BSN2.IN.Tact )
      Coil( #TS_StationBSN2.EndOfCycle )
   END_RUNG
   // the same network as SCL:
   #TS_StationBSN2.EndOfCycle := NOT "Communication".BSN2.IN.Tact;
END_REGION

REGION Network 230: Station BSN2 - End of production
   RUNG wire#powerrail
      { S7_Templates := "SrcType := Int" } EQ_Contact(in1 := "STATUS_BSN2".Device.Specific.ConvPartCnt, in2 := 0)
      { S7_Templates := "SrcType := Int" } EQ_Contact(in1 := "STATUS_BSN2".Device.Specific.FurnacePartCnt, in2 := 0)
      wire#w1
      Coil( #TS_StationBSN2.EndOfProd )
   END_RUNG
   RUNG wire#powerrail
      Contact( "JKU1Comm" )
   END_RUNG wire#w1
   // the same network as SCL:
   #TS_StationBSN2.EndOfProd := (("STATUS_BSN2".Device.Specific.ConvPartCnt = 0) AND ("STATUS_BSN2".Device.Specific.FurnacePartCnt = 0)) OR "JKU1Comm";
END_REGION

REGION Network 231: Station BSN2 - Main control
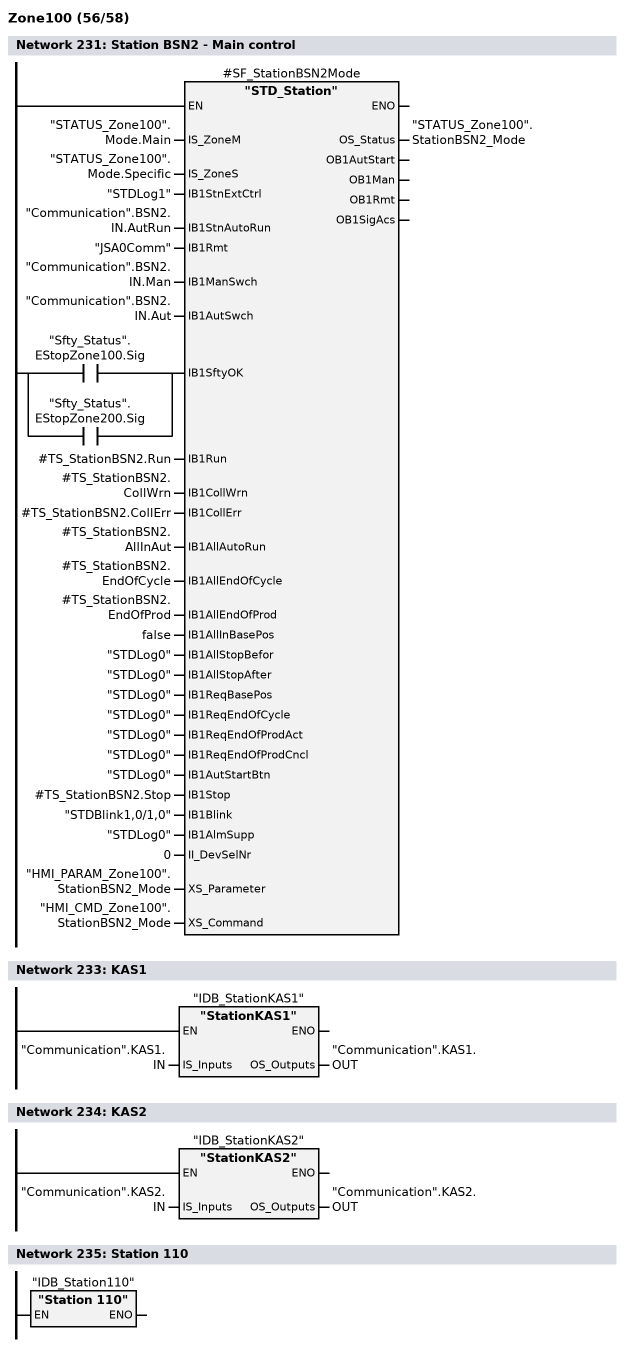
   RUNG wire#powerrail
      #SF_StationBSN2Mode(IB1SftyOK := wire#w1, IS_ZoneM := "STATUS_Zone100".Mode.Main, IS_ZoneS := "STATUS_Zone100".Mode.Specific, IB1StnExtCtrl := "STDLog1", IB1StnAutoRun := "Communication".BSN2.IN.AutRun, IB1Rmt := "JSA0Comm", IB1ManSwch := "Communication".BSN2.IN.Man, IB1AutSwch := "Communication".BSN2.IN.Aut, IB1Run := #TS_StationBSN2.Run, IB1CollWrn := #TS_StationBSN2.CollWrn, IB1CollErr := #TS_StationBSN2.CollErr, IB1AllAutoRun := #TS_StationBSN2.AllInAut, IB1AllEndOfCycle := #TS_StationBSN2.EndOfCycle, IB1AllEndOfProd := #TS_StationBSN2.EndOfProd, IB1AllInBasePos := false, IB1AllStopBefor := "STDLog0", IB1AllStopAfter := "STDLog0", IB1ReqBasePos := "STDLog0", IB1ReqEndOfCycle := "STDLog0", IB1ReqEndOfProdAct := "STDLog0", IB1ReqEndOfProdCncl := "STDLog0", IB1AutStartBtn := "STDLog0", IB1Stop := #TS_StationBSN2.Stop, IB1Blink := "STDBlink1,0/1,0", IB1AlmSupp := "STDLog0", II_DevSelNr := 0, XS_Parameter := "HMI_PARAM_Zone100".StationBSN2_Mode, XS_Command := "HMI_CMD_Zone100".StationBSN2_Mode, OS_Status => "STATUS_Zone100".StationBSN2_Mode, OB1AutStart =>, OB1Man =>, OB1Rmt =>, OB1SigAcs =>)
   END_RUNG
   RUNG wire#powerrail
      Contact( "Sfty_Status".EStopZone100.Sig )
   END_RUNG wire#w1
   RUNG wire#powerrail
      Contact( "Sfty_Status".EStopZone200.Sig )
   END_RUNG wire#w1
   // the same network as SCL:
   #SF_StationBSN2Mode(IS_ZoneM := "STATUS_Zone100".Mode.Main,   // "STD_Station"
                       IS_ZoneS := "STATUS_Zone100".Mode.Specific,
                       IB1StnExtCtrl := "STDLog1",
                       IB1StnAutoRun := "Communication".BSN2.IN.AutRun,
                       IB1Rmt := "JSA0Comm",
                       IB1ManSwch := "Communication".BSN2.IN.Man,
                       IB1AutSwch := "Communication".BSN2.IN.Aut,
                       IB1SftyOK := "Sfty_Status".EStopZone100.Sig OR "Sfty_Status".EStopZone200.Sig,
                       IB1Run := #TS_StationBSN2.Run,
                       IB1CollWrn := #TS_StationBSN2.CollWrn,
                       IB1CollErr := #TS_StationBSN2.CollErr,
                       IB1AllAutoRun := #TS_StationBSN2.AllInAut,
                       IB1AllEndOfCycle := #TS_StationBSN2.EndOfCycle,
                       IB1AllEndOfProd := #TS_StationBSN2.EndOfProd,
                       IB1AllInBasePos := false,
                       IB1AllStopBefor := "STDLog0",
                       IB1AllStopAfter := "STDLog0",
                       IB1ReqBasePos := "STDLog0",
                       IB1ReqEndOfCycle := "STDLog0",
                       IB1ReqEndOfProdAct := "STDLog0",
                       IB1ReqEndOfProdCncl := "STDLog0",
                       IB1AutStartBtn := "STDLog0",
                       IB1Stop := #TS_StationBSN2.Stop,
                       IB1Blink := "STDBlink1,0/1,0",
                       IB1AlmSupp := "STDLog0",
                       II_DevSelNr := 0,
                       XS_Parameter := "HMI_PARAM_Zone100".StationBSN2_Mode,
                       XS_Command := "HMI_CMD_Zone100".StationBSN2_Mode,
                       OS_Status => "STATUS_Zone100".StationBSN2_Mode);
END_REGION

REGION Network 232: *************** Call of stations ***************
END_REGION

REGION Network 233: KAS1
   RUNG wire#powerrail
      "IDB_StationKAS1"(IS_Inputs := "Communication".KAS1.IN, OS_Outputs => "Communication".KAS1.OUT)
   END_RUNG
   // the same network as SCL:
   "IDB_StationKAS1"(IS_Inputs := "Communication".KAS1.IN, OS_Outputs => "Communication".KAS1.OUT);   // "StationKAS1"
END_REGION

REGION Network 234: KAS2
   RUNG wire#powerrail
      "IDB_StationKAS2"(IS_Inputs := "Communication".KAS2.IN, OS_Outputs => "Communication".KAS2.OUT)
   END_RUNG
   // the same network as SCL:
   "IDB_StationKAS2"(IS_Inputs := "Communication".KAS2.IN, OS_Outputs => "Communication".KAS2.OUT);   // "StationKAS2"
END_REGION

REGION Network 235: Station 110
   RUNG wire#powerrail
      "IDB_Station110"()
   END_RUNG
   // the same network as SCL:
   "IDB_Station110"();   // "Station 110"
END_REGION

REGION Network 236: Station 120
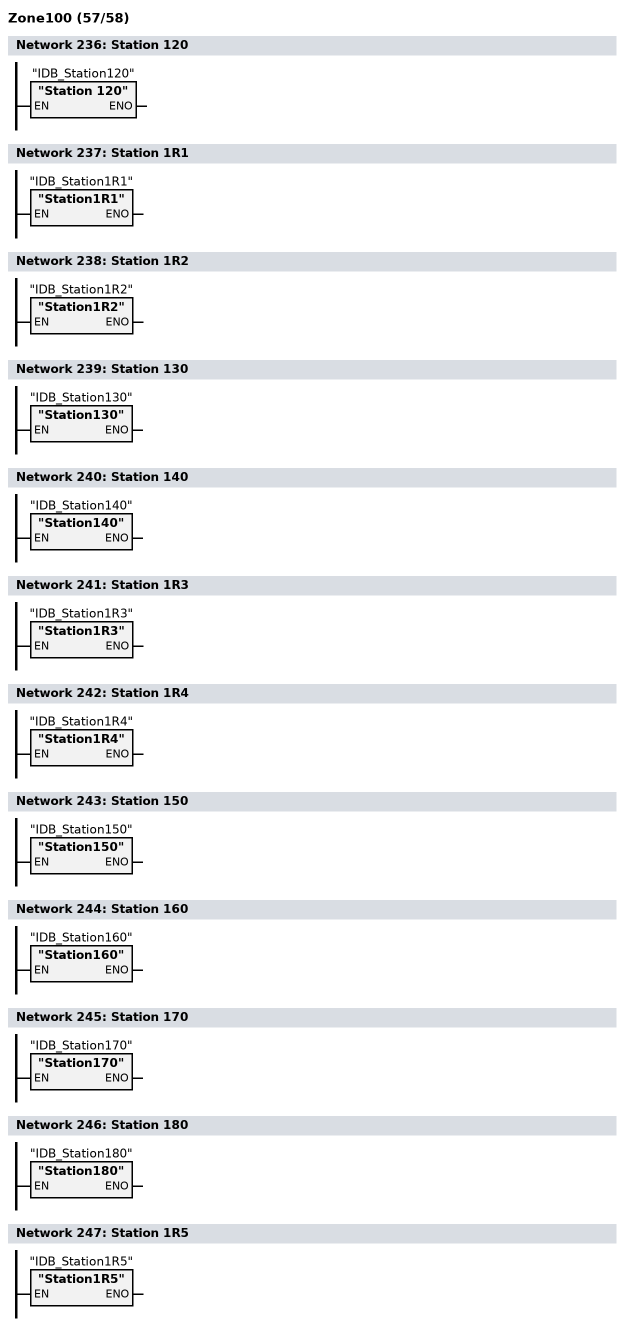
   RUNG wire#powerrail
      "IDB_Station120"()
   END_RUNG
   // the same network as SCL:
   "IDB_Station120"();   // "Station 120"
END_REGION

REGION Network 237: Station 1R1
   RUNG wire#powerrail
      "IDB_Station1R1"()
   END_RUNG
   // the same network as SCL:
   "IDB_Station1R1"();   // "Station1R1"
END_REGION

REGION Network 238: Station 1R2
   RUNG wire#powerrail
      "IDB_Station1R2"()
   END_RUNG
   // the same network as SCL:
   "IDB_Station1R2"();   // "Station1R2"
END_REGION

REGION Network 239: Station 130
   RUNG wire#powerrail
      "IDB_Station130"()
   END_RUNG
   // the same network as SCL:
   "IDB_Station130"();   // "Station130"
END_REGION

REGION Network 240: Station 140
   RUNG wire#powerrail
      "IDB_Station140"()
   END_RUNG
   // the same network as SCL:
   "IDB_Station140"();   // "Station140"
END_REGION

REGION Network 241: Station 1R3
   RUNG wire#powerrail
      "IDB_Station1R3"()
   END_RUNG
   // the same network as SCL:
   "IDB_Station1R3"();   // "Station1R3"
END_REGION

REGION Network 242: Station 1R4
   RUNG wire#powerrail
      "IDB_Station1R4"()
   END_RUNG
   // the same network as SCL:
   "IDB_Station1R4"();   // "Station1R4"
END_REGION

REGION Network 243: Station 150
   RUNG wire#powerrail
      "IDB_Station150"()
   END_RUNG
   // the same network as SCL:
   "IDB_Station150"();   // "Station150"
END_REGION

REGION Network 244: Station 160
   RUNG wire#powerrail
      "IDB_Station160"()
   END_RUNG
   // the same network as SCL:
   "IDB_Station160"();   // "Station160"
END_REGION

REGION Network 245: Station 170
   RUNG wire#powerrail
      "IDB_Station170"()
   END_RUNG
   // the same network as SCL:
   "IDB_Station170"();   // "Station170"
END_REGION

REGION Network 246: Station 180
   RUNG wire#powerrail
      "IDB_Station180"()
   END_RUNG
   // the same network as SCL:
   "IDB_Station180"();   // "Station180"
END_REGION

REGION Network 247: Station 1R5
   RUNG wire#powerrail
      "IDB_Station1R5"()
   END_RUNG
   // the same network as SCL:
   "IDB_Station1R5"();   // "Station1R5"
END_REGION

REGION Network 248: Station 1R6
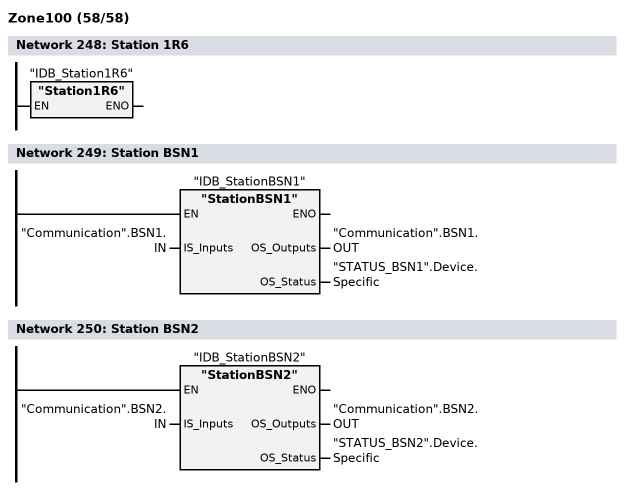
   RUNG wire#powerrail
      "IDB_Station1R6"()
   END_RUNG
   // the same network as SCL:
   "IDB_Station1R6"();   // "Station1R6"
END_REGION

REGION Network 249: Station BSN1
   RUNG wire#powerrail
      "IDB_StationBSN1"(IS_Inputs := "Communication".BSN1.IN, OS_Outputs => "Communication".BSN1.OUT, OS_Status => "STATUS_BSN1".Device.Specific)
   END_RUNG
   // the same network as SCL:
   "IDB_StationBSN1"(IS_Inputs := "Communication".BSN1.IN,   // "StationBSN1"
                     OS_Outputs => "Communication".BSN1.OUT,
                     OS_Status => "STATUS_BSN1".Device.Specific);
END_REGION

REGION Network 250: Station BSN2
   RUNG wire#powerrail
      "IDB_StationBSN2"(IS_Inputs := "Communication".BSN2.IN, OS_Outputs => "Communication".BSN2.OUT, OS_Status => "STATUS_BSN2".Device.Specific)
   END_RUNG
   // the same network as SCL:
   "IDB_StationBSN2"(IS_Inputs := "Communication".BSN2.IN,   // "StationBSN2"
                     OS_Outputs => "Communication".BSN2.OUT,
                     OS_Status => "STATUS_BSN2".Device.Specific);
END_REGION
END_FUNCTION_BLOCK
